# EPICS IOC start-up script: examples/test/elm7222/startup_ch1.iocsh
require ecmccfg, "ENG_MODE=1"

${SCRIPTEXEC} ${ECMC_CONFIG_ROOT}addSlave.cmd,      "HW_DESC=ELM7222-0010, SLAVE_ID=21"
${SCRIPTEXEC} ${ecmccfg_DIR}applySlaveConfig.cmd,   "CONFIG=-Motor-ch1-Beckhoff-AM8112-xFx1"

epicsEnvSet("DRV_SLAVE", ${ECMC_EC_SLAVE_NUM})
${SCRIPTEXEC} ${ECMC_CONFIG_ROOT}loadYamlAxis.cmd,  "FILE=cfg/AM8112_ch1.yaml, DEV=${DEV=${IOC}}, DRV_SLAVE=${DRV_SLAVE}"

#- #############################################################################
#- apply configuration
${SCRIPTEXEC} ${ECMC_CONFIG_ROOT}applyConfig.cmd
#- #############################################################################
#- go active
${SCRIPTEXEC} ${ECMC_CONFIG_ROOT}setAppMode.cmd

#- be quiet
asynSetTraceMask(MC_CPU1, -1, 0x01)
asynSetTraceIOMask(MC_CPU1, -1, 6)
asynSetTraceInfoMask(MC_CPU1, -1, 1)

#- reset all errors
ecmcConfigOrDie "ControllerErrorReset()"
